RoboDK station: kr30 cnc template in progress.rdk

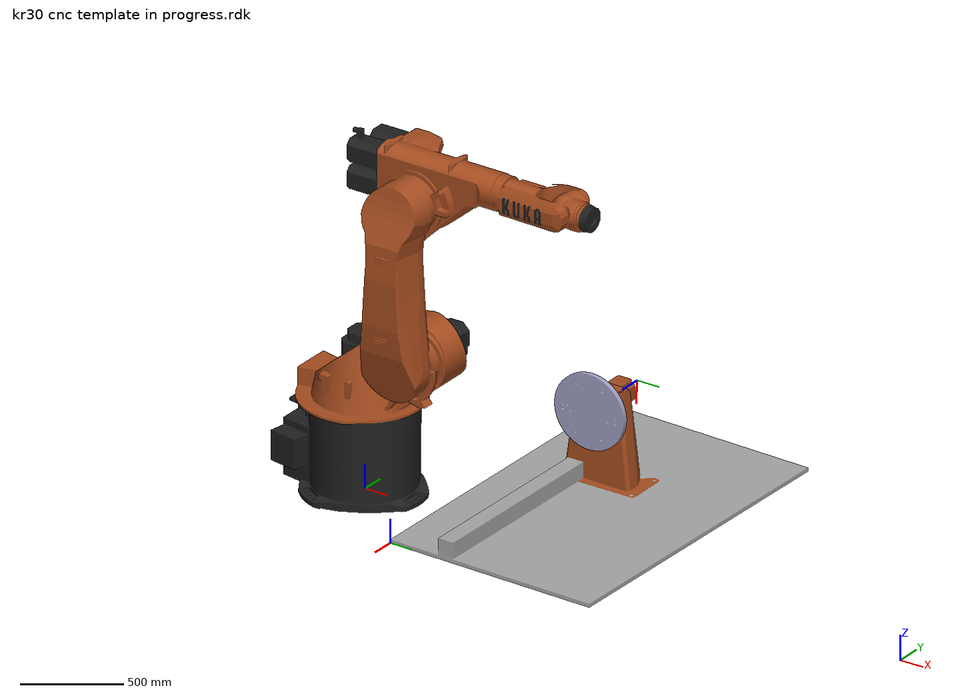
[picture v0: the station drawn from its stored meshes, robots at their saved joint values, targets as dots, program paths as lines]
Station kr30 cnc template in progress. Poses are relative to the parent item; angles as X-Y-Z fixed-axis rotations.
  - frame KUKA KR 30 HA Base at (0, 0, 0) mm
    - robot KUKA KR 30 HA: 6 axes, payload 30 kg, reach 2033 mm, repeatability 0.05 mm, weight 665 kg
        modified DH rows (alpha deg, a mm, theta deg, d mm): 0, 0, 0, 815; -90, 350, 0, 0; 0, 850, -90, 0; -90, 145, 0, 820; 90, 0, 0, 0; -90, 0, 180, 170
        joint limits [-185, -135, -120, -350, -119, -350] to [185, 35, 158, 350, 119, 350]; home [0, -90, 90, 0, 0, 0]; saved at [0, -90, 90, 0, 0, 0]
      - tool Tool 2, TCP at (337.71, -2.2, 160.57) mm, rotated rx 0 ry 90 rz 0 deg
    - frame Tabletop at (921.82, -1104.91, 407.05) mm, rotated rx -0.93 ry -0.21 rz -89.9 deg
      - object tabletop CHECK HEIGHT at (-1839.9, 0, 0) mm, size 1839.9 x 1168.4 x 19 mm, geometry from kr30 tabletop mm.stl
      - object kr30 pipe jig base at (-1220, -610.6, 0) mm, size 1217.6 x 88.9 x 88.9 mm, geometry from kr30 pipe jig base.stl
      - frame KUKA KP1 MD250 Base at (-1441.97, 434.54, 429.83) mm, rotated rx -120.7 ry 89.48 rz -119.27 deg
        - robot KUKA KP1 MD250: 1 axes, payload 250 kg
            modified DH rows (alpha deg, a mm, theta deg, d mm): 0, 0, 0, 0
            base shift (0, 0, 420) mm
            joint limits [-180] to [180]; home [0]; saved at [0]
